(* CoDeSys 2.3 export: PLC_PRG.EXP *)

(* POU PLC_PRG, ST *)
PROGRAM PLC_PRG
VAR
END_VAR
ClockCycles();
OptimizedTimer();
PC20_CYCLE();
IO_Mapping();
END_PROGRAM
